SYSTEM Stream
  (* Version 1.0, 2023-01-25, obotnar *)
  APPLICATION StreamApp
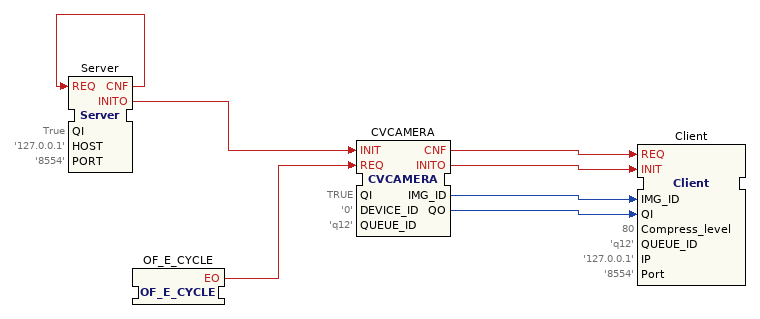
    FBS
      Server : Server(QI := True, HOST := '127.0.0.1', PORT := '8554');
      Client : Client(Compress_level := 80, QUEUE_ID := 'q12', IP := '127.0.0.1', Port := '8554');
      CVCAMERA : CVCAMERA(QI := TRUE, DEVICE_ID := '0', QUEUE_ID := 'q12');
      OF_E_CYCLE : OF_E_CYCLE;
    END_FBS
    EVENT_CONNECTIONS
      Server.CNF TO Server.REQ;
      Server.INITO TO CVCAMERA.INIT;
      CVCAMERA.CNF TO Client.REQ;
      CVCAMERA.INITO TO Client.INIT;
      OF_E_CYCLE.EO TO CVCAMERA.REQ;
    END_CONNECTIONS
    DATA_CONNECTIONS
      CVCAMERA.IMG_ID TO Client.IMG_ID;
      CVCAMERA.QO TO Client.QI;
    END_CONNECTIONS
  END_APPLICATION
  DEVICE FORTE_PC : FORTE_PC(MGR_ID := "10.5.20.122:61499" (* Device manager socket ID *))
    {SET_ATTRIBUTE(Profile, HOLOBLOC)}
    RESOURCE EMB_RES : 
    END_RESOURCE
  END_DEVICE
  MAPPINGS
    StreamApp.Server ON FORTE_PC.EMB_RES;
    StreamApp.Client ON FORTE_PC.EMB_RES;
    StreamApp.CVCAMERA ON FORTE_PC.EMB_RES;
    StreamApp.OF_E_CYCLE ON FORTE_PC.EMB_RES;
  END_MAPPINGS
  SEGMENTS
    Ethernet : Ethernet;
  END_SEGMENTS
  LINKS
    FORTE_PC => Ethernet;
  END_LINKS
END_SYSTEM
